(* PLC project BasicProgramTemplate, Industrial AI Agent CODESYS 3.5.21.0 *)
(* stored: creationDateTime 2026-06-10T10:00:00, modificationDateTime 2026-06-10T10:00:00 *)

PROGRAM PLC_PRG
  VAR
    xRun : BOOL;  (* Program calisma bayragi *)
    iCounter : INT := 0;
    rValue : REAL := 0.0;
  END_VAR

                        
// ------------------------------------------------------------
// PLC_PRG - Temel program sablonu
// Her cevrimde sayaci artirir ve basit bir hesaplama yapar.
// ------------------------------------------------------------

xRun := TRUE;

IF xRun THEN
    iCounter := iCounter + 1;

    // 1000'e ulasinca basa don
    IF iCounter >= 1000 THEN
        iCounter := 0;
    END_IF

    // Ornek hesaplama
    rValue := INT_TO_REAL(iCounter) * 0.1;
END_IF

                    
END_PROGRAM
